PROGRAM P4_03_Export
VAR
	fbExportAudit					:FB_PythonScript;
END_VAR

VAR PERSISTENT
	sLastExportedAuditTime			:STRING;
	sLastExportedAuditName			:STRING;
END_VAR
VAR // added by the converter: edge detectors and wires of the graphical bodies
    _rt1, _rt2 : R_TRIG;
END_VAR

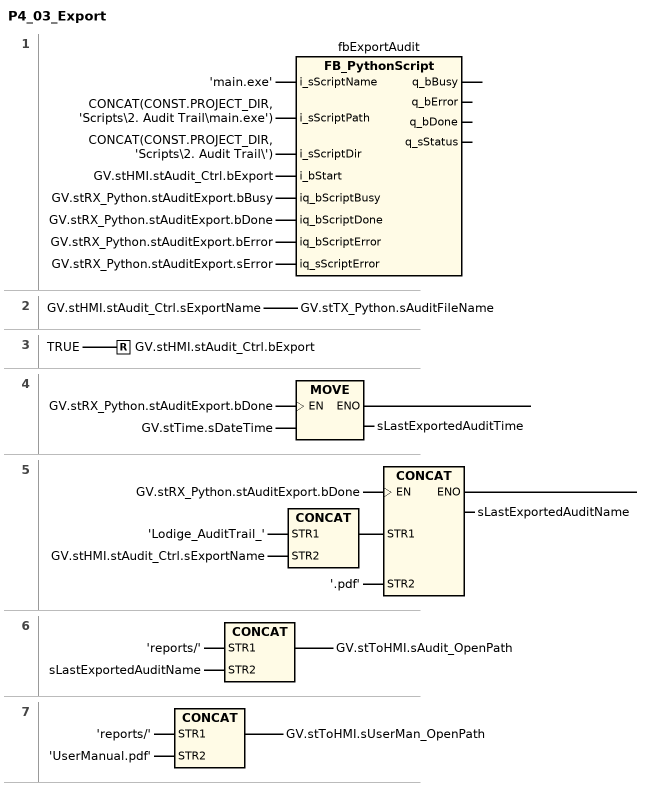
// NETWORK 1
fbExportAudit(
    i_sScriptName := 'main.exe',
    i_sScriptPath := CONCAT(CONST.PROJECT_DIR,'Scripts\2. Audit Trail\main.exe'),
    i_sScriptDir := CONCAT(CONST.PROJECT_DIR,'Scripts\2. Audit Trail\'),
    i_bStart := GV.stHMI.stAudit_Ctrl.bExport,
    iq_bScriptBusy := GV.stRX_Python.stAuditExport.bBusy,
    iq_bScriptDone := GV.stRX_Python.stAuditExport.bDone,
    iq_bScriptError := GV.stRX_Python.stAuditExport.bError,
    iq_sScriptError := GV.stRX_Python.stAuditExport.sError); // FB_PythonScript

// NETWORK 2
GV.stTX_Python.sAuditFileName := GV.stHMI.stAudit_Ctrl.sExportName;

// NETWORK 3
GV.stHMI.stAudit_Ctrl.bExport R= TRUE;

// NETWORK 4
_rt1(CLK := GV.stRX_Python.stAuditExport.bDone);
IF _rt1.Q THEN sLastExportedAuditTime := GV.stTime.sDateTime; END_IF

// NETWORK 5
_rt2(CLK := GV.stRX_Python.stAuditExport.bDone);
IF _rt2.Q THEN
    sLastExportedAuditName := CONCAT(STR1 := CONCAT(STR1 := 'Lodige_AuditTrail_', STR2 := GV.stHMI.stAudit_Ctrl.sExportName), STR2 := '.pdf');
END_IF

// NETWORK 6
GV.stToHMI.sAudit_OpenPath := CONCAT(STR1 := 'reports/', STR2 := sLastExportedAuditName);

// NETWORK 7
GV.stToHMI.sUserMan_OpenPath := CONCAT(STR1 := 'reports/', STR2 := 'UserManual.pdf');

END_PROGRAM

(* stored: Version 1.1.0.1
   POU P4_03_Export: Id {6f3bd936-e46b-4e39-b559-4f72aa8a5abe}, SpecialFunc None *)
